// TIA Portal project "Çevrimsel_Kesme_Uygulaması_V1" (V16)
// Vorlageprojekt für das Buch mit Zielsystem S7-1200

(* hardware
DEVICE "S7-1200-Station_1"  S7-1200 Station
   slot 0: "Baugruppenträger_0"  Rack  V1.0
   slot 1: "PLC_1"  CPU 1214C DC/DC/DC  6ES7 214-1AG40-0XB0  V4.4
   slot 2: "AQ 4x14BIT_1"  6ES7 232-4HD32-0XB0  V2.1
*)

// ===== PLC "PLC_1"  CPU 1214C DC/DC/DC =====

VAR_GLOBAL   // PLC tag table "Standard-Variablentabelle"
   "Sitem_Start_Mem" AT %M10.0 : Bool;
   "Sıvı_Seviyesi_1" AT %MD20 : Real;
   "Sıvı_Seviyesi_2" AT %MD24 : Real;
   "Tank_Dolu_Mem." AT %M11.0 : Bool;
   "Kesme_Sinyali" AT %M30.0 : Bool;
END_VAR

VAR_GLOBAL   // PLC tag table "Input"
   "Start_But" AT %I0.0 : Bool;
   "Stop_But" AT %I0.1 : Bool;
   "Seviye_Tespit_Sensörü_1" AT %IW30 : Int;
   "Seviye_Tespit_Sensörü_2" AT %IW32 : Int;
END_VAR

VAR_GLOBAL   // PLC tag table "Output"
   "Sinyal_Lambası" AT %Q0.0 : Bool;
   "Doldurma_Valfi_2" AT %QW30 : Int;
   "Doldurma_Valfi_1" AT %QW32 : Int;
   "Boşaltma_Valfi_1" AT %QW34 : Int;
   "Boşaltma_Valfi_2" AT %QW36 : Int;
END_VAR

DATA_BLOCK "Tank_Seviye_1"   // DB1
{ S7_Optimized_Access := 'TRUE' }
VERSION : 0.1
// stored: InstanceOfName Sıvı Seviyesini Okuma
"Sıvı Seviyesini Okuma"
BEGIN
END_DATA_BLOCK

DATA_BLOCK "Tank_Seviye_2"   // DB2
{ S7_Optimized_Access := 'TRUE' }
VERSION : 0.1
// stored: InstanceOfName Sıvı Seviyesini Okuma
"Sıvı Seviyesini Okuma"
BEGIN
END_DATA_BLOCK

FUNCTION_BLOCK "Sıvı Seviyesini Okuma"   // FB1, LAD
{ S7_Optimized_Access := 'TRUE' }
VERSION : 0.1
   VAR_INPUT
      Sıvı_Seviye_Sensörü_Girişi : Int;
   END_VAR
   VAR_OUTPUT
      Sıvı_Seviyesi : Real;
   END_VAR
   VAR
      Marker_1 : Int;
      Marker_2 : Real;
   END_VAR
BEGIN

REGION Network 1: Sıvı Seviyesini Okuma 1
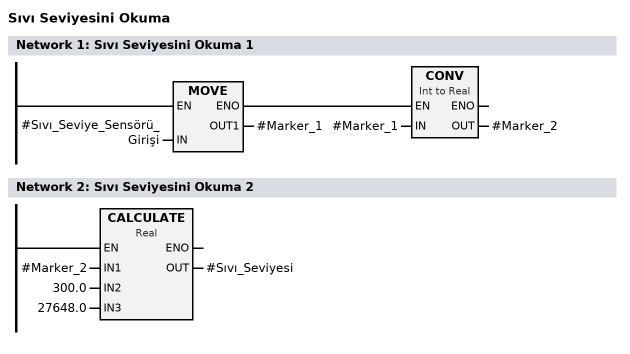
   RUNG wire#powerrail
      Move(in := #Sıvı_Seviye_Sensörü_Girişi, out1 => #Marker_1)
      { S7_Templates := "[SrcType := Int, DestType := Real]" } Convert(in := #Marker_1, out => #Marker_2)
   END_RUNG
   // the same network as SCL:
   #Marker_1 := #Sıvı_Seviye_Sensörü_Girişi;
   #Marker_2 := INT_TO_REAL(#Marker_1);
END_REGION

REGION Network 2: Sıvı Seviyesini Okuma 2
   RUNG wire#powerrail
      { S7_Templates := "SrcType := Real"; S7_Expression := "(IN1 * IN2) /IN3" } Calculate(in1 := #Marker_2, in2 := 300.0, in3 := 27648.0, out => #Sıvı_Seviyesi)
   END_RUNG
   // the same network as SCL:
   #Sıvı_Seviyesi := (#Marker_2 * 300.0) /27648.0;
END_REGION
END_FUNCTION_BLOCK

FUNCTION "MHJ-PLC-Lab-Function-S71200" : Void   // FC9000, SCL
{ S7_Optimized_Access := 'TRUE' }
VERSION : 0.1
   VAR_TEMP
      rdTimeReturn : Int;
      outputTime : DTL;
      SyncVal : Byte;
      forVal : Int;
      forVal_2 : Int;
      Value : Byte;
   END_VAR
   VAR CONSTANT
      CompVal : Byte := 16#34;
      Value_01 : Byte := 16#11;
      Value_01_DW : DWord := 16#A165_D992;
      Value_02_DW : DWord := 16#58BE_4401;
   END_VAR
BEGIN

   #Value:=PEEK(area := 16#82,
        dbNumber := 0,
        byteOffset := 511);
   #Value := #Value + 1;

   POKE(area := 16#82,
        dbNumber := 0,
        byteOffset := 511,
        value := #Value);

   POKE(area:=16#81,
        dbNumber:=0,
        byteOffset:=1016,
        value:=#Value_01_DW);
   POKE(area := 16#81,
        dbNumber := 0,
        byteOffset := 1020,
        value := #Value_02_DW);

   POKE(area := 16#81,
        dbNumber := 0,
        byteOffset := 511,
        value := B#16#00);

   FOR #forVal := 0 TO 120 DO
       FOR #forVal_2:=0 TO 10 DO
           #rdTimeReturn:=RD_SYS_T(#outputTime);
           #rdTimeReturn := WR_SYS_T(#outputTime);
           #rdTimeReturn := RD_SYS_T(#outputTime);
           #rdTimeReturn := WR_SYS_T(#outputTime);
       END_FOR;
       #SyncVal:= PEEK(area := 16#81,
                      dbNumber := 0,
                      byteOffset := 511);
       IF #SyncVal = #CompVal THEN
          GOTO M_1;
       END_IF;
   END_FOR;
   RETURN;

   M_1:
   POKE(area := 16#81,
        dbNumber := 0,
        byteOffset := 511,
        value := B#16#0);
END_FUNCTION

ORGANIZATION_BLOCK "Main"   // OB1, LAD, ProgramCycle
TITLE = "Main Program Sweep (Cycle)"
{ S7_Optimized_Access := 'TRUE' }
VERSION : 0.1
   VAR_INPUT
      Initial_Call : Bool;   // Initial call of this OB
      Remanence : Bool;   // =True, if remanent data are available
   END_VAR
   VAR_TEMP   // added for the SCL form of the ladder/FBD networks
      _w1 : Bool;
   END_VAR
BEGIN

REGION Network 1: Konnektierungsbaustein für PLC-Lab
   // Im Netzwerk 1 wird der Konnektierungsbaustein für PLC-Lab aufgerufen.
   // Dieser Aufruf darf nicht entfernt werden!
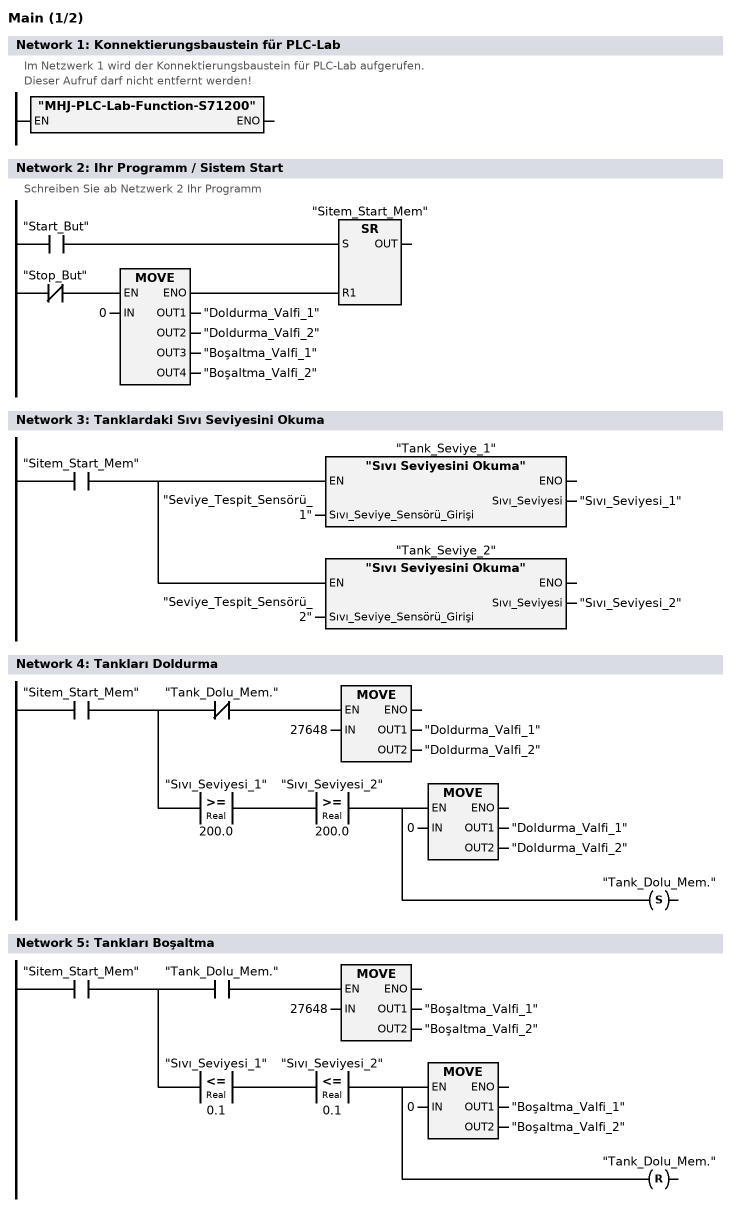
   RUNG wire#powerrail
      "MHJ-PLC-Lab-Function-S71200"()
   END_RUNG
   // the same network as SCL:
   "MHJ-PLC-Lab-Function-S71200"();
END_REGION

REGION Network 2: Ihr Programm / Sistem Start
   // Schreiben Sie ab Netzwerk 2 Ihr Programm
   RUNG wire#powerrail
      Contact( "Start_But" )
      S_SR(operand := "Sitem_Start_Mem", r1 := wire#w1)
   END_RUNG
   RUNG wire#powerrail
      I_Contact( "Stop_But" )
      Move(in := 0, out1 => "Doldurma_Valfi_1", out2 => "Doldurma_Valfi_2", out3 => "Boşaltma_Valfi_1", out4 => "Boşaltma_Valfi_2")
   END_RUNG wire#w1
   // the same network as SCL:
   IF NOT "Stop_But" THEN
       "Doldurma_Valfi_1" := 0;
       "Doldurma_Valfi_2" := 0;
       "Boşaltma_Valfi_1" := 0;
       "Boşaltma_Valfi_2" := 0;
   END_IF;
   IF "Start_But" THEN
       "Sitem_Start_Mem" := TRUE;   // SR flip-flop
   END_IF;
   IF NOT "Stop_But" THEN "Sitem_Start_Mem" := FALSE; END_IF;
END_REGION

REGION Network 3: Tanklardaki Sıvı Seviyesini Okuma
   RUNG wire#powerrail
      Contact( "Sitem_Start_Mem" )
      wire#w1
      "Tank_Seviye_1"(Sıvı_Seviye_Sensörü_Girişi := "Seviye_Tespit_Sensörü_1", Sıvı_Seviyesi => "Sıvı_Seviyesi_1")
   END_RUNG
   RUNG wire#w1
      "Tank_Seviye_2"(Sıvı_Seviye_Sensörü_Girişi := "Seviye_Tespit_Sensörü_2", Sıvı_Seviyesi => "Sıvı_Seviyesi_2")
   END_RUNG
   // the same network as SCL:
   #_w1 := "Sitem_Start_Mem";
   IF #_w1 THEN
       "Tank_Seviye_1"(Sıvı_Seviye_Sensörü_Girişi := "Seviye_Tespit_Sensörü_1", Sıvı_Seviyesi => "Sıvı_Seviyesi_1");   // "Sıvı Seviyesini Okuma"
       "Tank_Seviye_2"(Sıvı_Seviye_Sensörü_Girişi := "Seviye_Tespit_Sensörü_2", Sıvı_Seviyesi => "Sıvı_Seviyesi_2");   // "Sıvı Seviyesini Okuma"
   END_IF;
END_REGION

REGION Network 4: Tankları Doldurma
   RUNG wire#powerrail
      Contact( "Sitem_Start_Mem" )
      wire#w1
      I_Contact( "Tank_Dolu_Mem." )
      Move(in := 27648, out1 => "Doldurma_Valfi_1", out2 => "Doldurma_Valfi_2")
   END_RUNG
   RUNG wire#w1
      { S7_Templates := "SrcType := Real" } GE_Contact(in1 := "Sıvı_Seviyesi_1", in2 := 200.0)
      { S7_Templates := "SrcType := Real" } GE_Contact(in1 := "Sıvı_Seviyesi_2", in2 := 200.0)
      wire#w2
      Move(in := 0, out1 => "Doldurma_Valfi_1", out2 => "Doldurma_Valfi_2")
   END_RUNG
   RUNG wire#w2
      S_Coil( "Tank_Dolu_Mem." )
   END_RUNG
   // the same network as SCL:
   IF "Sitem_Start_Mem" AND NOT "Tank_Dolu_Mem." THEN
       "Doldurma_Valfi_1" := 27648;
       "Doldurma_Valfi_2" := 27648;
   END_IF;
   IF "Sitem_Start_Mem" AND ("Sıvı_Seviyesi_1" >= 200.0) AND ("Sıvı_Seviyesi_2" >= 200.0) THEN
       "Doldurma_Valfi_1" := 0;
       "Doldurma_Valfi_2" := 0;
       "Tank_Dolu_Mem." := TRUE;
   END_IF;
END_REGION

REGION Network 5: Tankları Boşaltma
   RUNG wire#powerrail
      Contact( "Sitem_Start_Mem" )
      wire#w1
      Contact( "Tank_Dolu_Mem." )
      Move(in := 27648, out1 => "Boşaltma_Valfi_1", out2 => "Boşaltma_Valfi_2")
   END_RUNG
   RUNG wire#w1
      { S7_Templates := "SrcType := Real" } LE_Contact(in1 := "Sıvı_Seviyesi_1", in2 := 0.1)
      { S7_Templates := "SrcType := Real" } LE_Contact(in1 := "Sıvı_Seviyesi_2", in2 := 0.1)
      wire#w2
      Move(in := 0, out1 => "Boşaltma_Valfi_1", out2 => "Boşaltma_Valfi_2")
   END_RUNG
   RUNG wire#w2
      R_Coil( "Tank_Dolu_Mem." )
   END_RUNG
   // the same network as SCL:
   IF "Sitem_Start_Mem" AND "Tank_Dolu_Mem." THEN
       "Boşaltma_Valfi_1" := 27648;
       "Boşaltma_Valfi_2" := 27648;
   END_IF;
   IF "Sitem_Start_Mem" AND ("Sıvı_Seviyesi_1" <= 0.1) AND ("Sıvı_Seviyesi_2" <= 0.1) THEN
       "Boşaltma_Valfi_1" := 0;
       "Boşaltma_Valfi_2" := 0;
       "Tank_Dolu_Mem." := FALSE;
   END_IF;
END_REGION

REGION Network 6: Kesme Sinyaline Göre Tankları Boşaltma
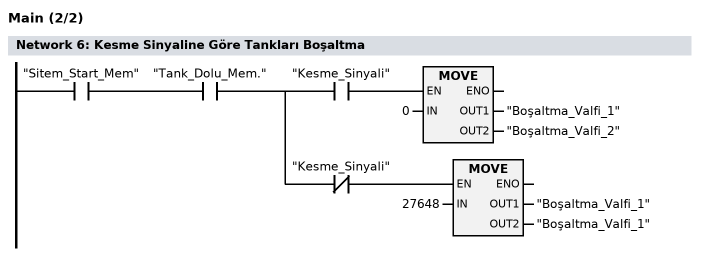
   RUNG wire#powerrail
      Contact( "Sitem_Start_Mem" )
      Contact( "Tank_Dolu_Mem." )
      wire#w1
      Contact( "Kesme_Sinyali" )
      Move(in := 0, out1 => "Boşaltma_Valfi_1", out2 => "Boşaltma_Valfi_2")
   END_RUNG
   RUNG wire#w1
      I_Contact( "Kesme_Sinyali" )
      Move(in := 27648, out1 => "Boşaltma_Valfi_1", out2 => "Boşaltma_Valfi_1")
   END_RUNG
   // the same network as SCL:
   #_w1 := "Sitem_Start_Mem" AND "Tank_Dolu_Mem.";
   IF #_w1 AND "Kesme_Sinyali" THEN
       "Boşaltma_Valfi_1" := 0;
       "Boşaltma_Valfi_2" := 0;
   END_IF;
   IF #_w1 AND NOT "Kesme_Sinyali" THEN
       "Boşaltma_Valfi_1" := 27648;
       "Boşaltma_Valfi_1" := 27648;
   END_IF;
END_REGION
END_ORGANIZATION_BLOCK

ORGANIZATION_BLOCK "Cyclic interrupt"   // OB30, LAD, CyclicInterrupt
{ S7_Optimized_Access := 'TRUE' }
VERSION : 0.1
   VAR_INPUT
      Initial_Call : Bool;   // Initial call of this OB
      Event_Count : Int;   // Events discarded
   END_VAR
BEGIN

REGION Network 1: Çevrimsel Kesme Sinyali
   // - Çevrimsel kesme, bir işlemin örneğin her 100 ms, 1 saniye veya 10 saniyede bir düzenli olarak çalıştırılmasını sağlar.
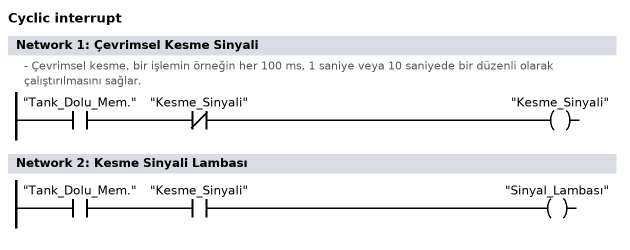
   RUNG wire#powerrail
      Contact( "Tank_Dolu_Mem." )
      I_Contact( "Kesme_Sinyali" )
      Coil( "Kesme_Sinyali" )
   END_RUNG
   // the same network as SCL:
   "Kesme_Sinyali" := "Tank_Dolu_Mem." AND NOT "Kesme_Sinyali";
END_REGION

REGION Network 2: Kesme Sinyali Lambası
   RUNG wire#powerrail
      Contact( "Tank_Dolu_Mem." )
      Contact( "Kesme_Sinyali" )
      Coil( "Sinyal_Lambası" )
   END_RUNG
   // the same network as SCL:
   "Sinyal_Lambası" := "Tank_Dolu_Mem." AND "Kesme_Sinyali";
END_REGION
END_ORGANIZATION_BLOCK